// TIA Portal V19 export
FUNCTION "FC_VAR_SPL" : Void   // FC13, STL
TITLE = Variable Sprungverteilung
{ S7_Optimized_Access := 'FALSE' }
AUTHOR : MS
// SPRUNGMARKENVORGABE FÜR VARIABLE SCHRITTFOLGEN
// stored: AutoNumber false
   VAR_INPUT
      Instanz_DB : Int;
   END_VAR
   VAR_OUTPUT
      Nr_MicroBef : Byte;
   END_VAR
   VAR_IN_OUT
      next_Step : Bool;
      Adr_MicroBef : Word;
   END_VAR
   VAR_TEMP
      FW_DB : DB_ANY;
      Adresse : DWord;
   END_VAR
BEGIN

NETWORK
TITLE = Programm
// Es ist ab einer festen Adresse des offenen DBs die Reihenfolge der 
// abzuarbeitenden Teilschritte einzugeben. (Schrittnummern der Größe Byte)
      L     #Instanz_DB;
      T     #FW_DB;
      OPN   DI [#FW_DB];

//BEI NEXT WIRD DIE JEWILIGE DB_ADR AKTIVIERT
//DIE SPRUNGADRESSE WIRD ÜBER STEP AUSGEGEBEN
      AN    #next_Step;
      AN    %DIX25.7;  //ZST.Start_UP
      R     %DIX25.2;  //neuer Befehl
      A     %DIX25.7;  //ZST.Start_UP
      JC    Init;
      AN    #next_Step;
      JC    Send;
      L     #Adr_MicroBef;
      L     1;
      +I;
      T     #Adr_MicroBef;
Init: S     %DIX25.2;  //neuer Befehl
      R     %DIX25.3;  //Befehls Merker
      R     %DIX25.4;  //Befehls Merker
      R     %DIX25.5;  //Befehls Merker
      R     %DIX25.6;  //Befehls Merker
      R     %DIX0.4;  //"DI_FW_1".ZST.HEBEN_AKT
      R     %DIX0.5;  //"DI_FW_1".ZST.SENKEN_AKT
      R     %DIX0.6;  //"DI_FW_1".ZST.VORWAERTS_AKT
      R     %DIX0.7;  //"DI_FW_1".ZST.RUECKWAERTS_AKT

Send: L     #Adr_MicroBef;
      SLD   3;
      T     #Adresse;
      L     DIB [#Adresse];
      T     #Nr_MicroBef;
      CLR;
      =     #next_Step;
      =     %DIX25.7;  //ZST.Start_UP
      BE;
END_FUNCTION
